Staubli VAL3: BackBoxType.pgx

public program BackBoxType()
begin
  if nBoxType>1
    nBoxType=nBoxType-1
  else
    nBoxType=2
  endIf
end
